TYPE ST_watertank_Input :
STRUCT
	In1: LREAL;
END_STRUCT
END_TYPE

(* stored: Version 1.1.0.1, ProductVersion 3.1.4024.4
   DUT ST_watertank_Input: Id {661db0d7-6076-4573-b23f-bb22e1647e83} *)
